TYPE ST_PML_Status :
STRUCT
    State : E_PML_State;
    Busy  : BOOL;
    Done  : BOOL;
    Error : BOOL;
    Info  : STRING(120);
END_STRUCT
END_TYPE

(* stored: Version 1.1.0.1, ProductVersion 3.1.4024.13
   DUT ST_PML_Status: Id {2d13f5ae-c731-4cd7-9ec2-cca80bbcb447} *)
